// TIA Portal V17 export
FUNCTION "移动指令_MOVE" : Void   // FC, LAD
{ S7_Optimized_Access := 'TRUE' }
VERSION : 0.1
// stored: AutoNumber true, IsIECCheckEnabled false, SetENOAutomatically false
BEGIN

REGION Network 1
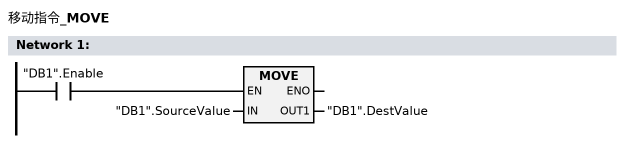
   RUNG wire#powerrail
      Contact( "DB1".Enable )
      { S7_GenerateENO := "TRUE" } Move(in := "DB1".SourceValue, out1 => "DB1".DestValue)
   END_RUNG
   // the same network as SCL:
   IF "DB1".Enable THEN "DB1".DestValue := "DB1".SourceValue; END_IF;
END_REGION
END_FUNCTION
